FUNCTION F_CommandAllSequences : BOOL
VAR_IN_OUT
	itfSequenceArray	: ARRAY[*] OF ITF_ModuleSequenceControl;
END_VAR
VAR_INPUT
	eCommand			: E_ModuleSequenceCommand;
	nSubCount			: UDINT;
END_VAR
VAR
	i:	UDINT;
END_VAR

CASE eCommand OF
	E_ModuleSequenceCommand.Clear:
		FOR i := 1 TO nSubCount DO
			itfSequenceArray[i].ClearSequence();
		END_FOR
		
	E_ModuleSequenceCommand.Disable:
		FOR i := 1 TO nSubCount DO
			itfSequenceArray[i].DisableSequence();
		END_FOR
	
	E_ModuleSequenceCommand.Enable:
		FOR i := 1 TO nSubCount DO
			itfSequenceArray[i].EnableSequence();
		END_FOR
	
	E_ModuleSequenceCommand.Reset:
		FOR i := 1 TO nSubCount DO
			itfSequenceArray[i].ResetSequence();
		END_FOR
	
	E_ModuleSequenceCommand.Resume:
		FOR i := 1 TO nSubCount DO
			itfSequenceArray[i].ResumeSequence();
		END_FOR
	
	E_ModuleSequenceCommand.Start:
		FOR i := 1 TO nSubCount DO
			itfSequenceArray[i].StartSequence();
		END_FOR
	
END_CASE

END_FUNCTION

(* stored: Version 1.1.0.1, ProductVersion 3.1.4024.9
   POU F_CommandAllSequences: Id {2a8ddc45-54b4-4d4f-af91-e4616bd76094}, SpecialFunc None *)
